TYPE ST_BaseLogger_HMI :
STRUCT
END_STRUCT
END_TYPE

(* stored: Version 1.1.0.1
   DUT ST_BaseLogger_HMI: Id {5fb8738b-690e-028a-35e6-f12e4079a5f0} *)
